FUNCTION_BLOCK ThreeConCtl (* Composite Function Block Type *)
  (* Standard: 61499-2 *)
  (* Version 0.2, 2003-12-05, JHC, Rockwell Automation, Renamed from NEWCOMPFB. *)
  (* Version 0.1, 2002-01-08, JHC, Rockwell Automation, Added DLY FB as example. *)
  (* Version 0.0, 2000-05-27, JHC, Rockwell Automation *)
  (* Compiler header: package fb.rt.cs725; *)
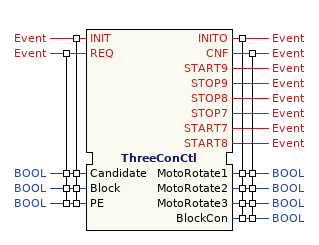
  EVENT_INPUT
    INIT WITH Candidate, Block, PE; (* Initialization Request *)
    REQ WITH Block, Candidate, PE; (* Normal Execution Request *)
  END_EVENT
  EVENT_OUTPUT
    INITO WITH MotoRotate1, MotoRotate2, MotoRotate3, BlockCon; (* Initialization Confirm *)
    CNF WITH MotoRotate1, MotoRotate2, MotoRotate3, BlockCon; (* Execution Confirmation *)
    START9;
    STOP9;
    STOP8;
    STOP7;
    START7;
    START8;
  END_EVENT
  VAR_INPUT
    Candidate : BOOL;
    Block : BOOL;
    PE : BOOL;
  END_VAR
  VAR_OUTPUT
    MotoRotate1 : BOOL;
    MotoRotate2 : BOOL;
    MotoRotate3 : BOOL;
    BlockCon : BOOL;
  END_VAR
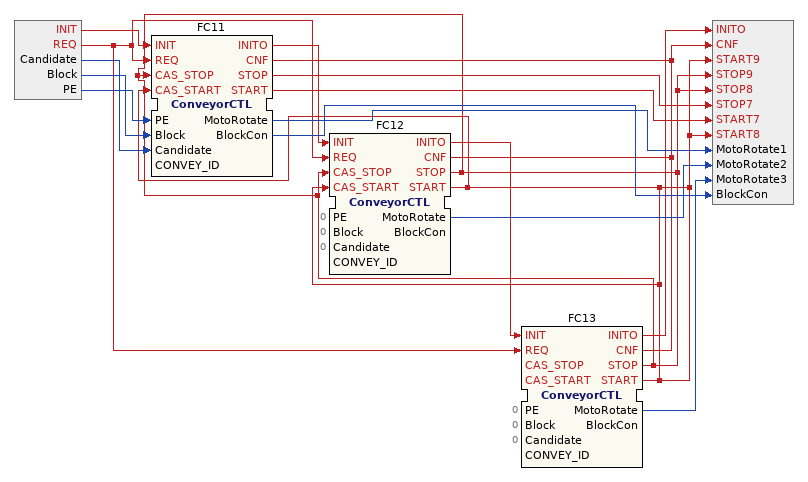
  FBS
    FC11 : ConveyorCTL;
    FC12 : ConveyorCTL(PE := 0, Block := 0, Candidate := 0);
    FC13 : ConveyorCTL(PE := 0, Block := 0, Candidate := 0);
  END_FBS
  EVENT_CONNECTIONS
    INIT TO FC11.INIT;
    REQ TO FC11.REQ;
    FC11.INITO TO FC12.INIT;
    FC12.INITO TO FC13.INIT;
    FC13.INITO TO INITO;
    FC13.CNF TO CNF;
    REQ TO FC12.REQ;
    REQ TO FC13.REQ;
    FC11.CNF TO CNF;
    FC12.CNF TO CNF;
    FC12.STOP TO STOP8;
    FC11.STOP TO STOP7;
    FC13.STOP TO STOP9;
    FC13.STOP TO FC11.CAS_STOP;
    FC13.STOP TO FC12.CAS_STOP;
    FC12.STOP TO FC11.CAS_STOP;
    FC13.START TO START9;
    FC11.START TO START7;
    FC12.START TO START8;
    FC12.START TO FC11.CAS_START;
    FC13.START TO FC11.CAS_START;
    FC13.START TO FC12.CAS_START;
  END_CONNECTIONS
  DATA_CONNECTIONS
    FC13.MotoRotate TO MotoRotate3;
    FC12.MotoRotate TO MotoRotate2;
    FC11.MotoRotate TO MotoRotate1;
    PE TO FC11.PE;
    Block TO FC11.Block;
    FC11.BlockCon TO BlockCon;
    Candidate TO FC11.Candidate;
  END_CONNECTIONS
END_FUNCTION_BLOCK
